FUNCTION_BLOCK FB2_Counters
VAR_INPUT
	ENable: Bool;
END_VAR
VAR_OUTPUT
END_VAR
VAR
END_VAR

VAR_STAT
	eenHzTrig: R_TRIG := FALSE;
END_VAR

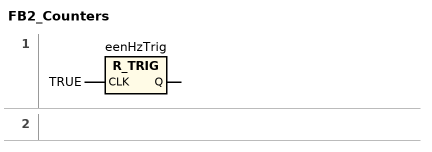
// NETWORK 1
eenHzTrig(CLK := TRUE); // R_TRIG

// NETWORK 2

END_FUNCTION_BLOCK

(* stored: Version 1.1.0.1, ProductVersion 3.1.4024.12
   POU FB2_Counters: Id {f4c5f6b3-94e5-44d7-9ae5-035ff107b3f1}, SpecialFunc None *)
